FUNCTION_BLOCK MC2_Axis_Base
VAR_INPUT
END_VAR
VAR_OUTPUT
END_VAR
VAR
	_axis : Tc2_MC2.AXIS_REF;
	axesEnable		: MC_Power;
	axesReset		: AxesReset(_axis);
	axesMoveTo 		: MoveSwitchToPosition(_axis);
	axesHalt 		: HaltMover(_axis);
	axesReadError : Tc2_MC2.MC_ReadAxisError;
	_MoverErrorId: DWORD;
END_VAR

axesMoveTo();
axesHalt();
axesReset();
_axis.ReadStatus();
axesEnable(Axis := _axis);
axesReadError(Axis := _axis, Enable := TRUE, AxisErrorID => _MoverErrorId);

METHOD PUBLIC DisableAxis : BOOL
VAR_INPUT
END_VAR
axesEnable.Enable := false;
END_METHOD

METHOD PUBLIC EnableAxis : BOOL
VAR_INPUT
END_VAR
axesEnable.Enable := axesEnable.Enable_Negative := axesEnable.Enable_Positive := TRUE;
axesEnable.Override := 100;
END_METHOD

METHOD PUBLIC HaltAxis : BOOL
VAR_INPUT
END_VAR
IF NOT axesHalt.Busy THEN
	axesHalt.Execute();
	HaltAxis := TRUE;
END_IF
END_METHOD

METHOD hasError : BOOL
VAR_INPUT
END_VAR
hasError := _axis.Status.Error;
END_METHOD

METHOD isAtPosition : BOOL
VAR_INPUT
	position : MC_LREAL;
END_VAR
IF _axis.NcToPlc.ModuloActPos < position + 0.2 AND _axis.NcToPlc.ModuloActPos > position - 0.2 THEN
	isAtPosition := TRUE;
END_IF
END_METHOD

METHOD isEnabled : BOOL
VAR_INPUT
END_VAR
isEnabled := not _axis.Status.Disabled;
END_METHOD

METHOD PUBLIC MoveTo : BOOL
VAR_INPUT
	Position : MC_LREAL;
	Velocity : MC_LREAL;
END_VAR
IF NOT isAtPosition(position := Position) THEN
	IF NOT axesMoveTo.Busy THEN
		axesMoveTo.MoveTo(Position := Position, Velocity := Velocity);
		MoveTo := TRUE;
	END_IF
END_IF
END_METHOD

END_FUNCTION_BLOCK

(* stored: Version 1.1.0.1, ProductVersion 3.1.4024.11
   POU MC2_Axis_Base: Id {ee6e7337-5f5f-4c5d-9917-89dff0d4a6cd}, SpecialFunc None
   Method DisableAxis: Id {dc075f9c-b535-4f77-a77b-3a861aeac30a}
   Method EnableAxis: Id {fd383078-082d-4269-8f8b-9ddb051d12fa}
   Method HaltAxis: Id {079fcc48-e6ef-4393-b619-932dde04fbb7}
   Method hasError: Id {e562e1dc-1d96-4854-a959-c047830f5072}
   Method isAtPosition: Id {759f3fe2-ecc3-47d7-a565-50175aea3510}
   Method isEnabled: Id {5aa08f06-f1a7-4864-95cb-b6f30feaf835}
   Method MoveTo: Id {10981345-e84c-491a-ba3f-6d3f1f0223b2} *)
